(* PLC project BE_Framework BA.project, CODESYS CODESYS V3.5 SP13 Patch 2 *)
(* stored: creationDateTime 2018-12-05T10:06:31.7537871, modificationDateTime 2018-12-03T08:58:43.5869763 *)

PROGRAM LB01_FF1_Analog
VAR
	local:strFan_Analog;
	localGP:strSensor2_Regulator;
	ControlFan: _BE_Fan;
	FbRegulator: _BE_Regulator;
	_BE_Fan2: _BE_Fan_2;
	reset_en: RS;
	AlarmFbAl01: _BE_AlarmAckRequired;
	AlarmFbAl02: _BE_AlarmAckRequired;
	fb_OperationalTime: _BE_OperationalTime;
	ackAl01: BOOL;
	ackAl02: BOOL;
	fanGuardOk: BOOL;
END_VAR
  VAR  (* added by the conversion: wires and edge detectors of the diagram *)
    __49_OUT : REAL;
    _MOVE171_ENO : BOOL;
    _MOVE171_OUT : INT;
    _AND235_OUT : BOOL;
    _AND241_OUT : BOOL;
    _MOVE64_ENO : BOOL;
    _MOVE64_OUT : REAL;
    _MOVE70_ENO : BOOL;
    _MOVE70_OUT : REAL;
    _MOVE151_ENO : BOOL;
    _MOVE151_OUT : ANY;
  END_VAR

(* CFC diagram, written out as Structured Text *)
(* Handling of enable and disable of regulator *)
local := LB01.FF1;
localGP := LB01.GP21;
fanGuardOk := LB01.GP23.V;
local.EnFeedbackError := >(local.SP4, 0);
local.EnThermalError := >(local.SP2, 0);
(* Feedback error *)
local.EnFanGuardError := >(local.SP3, 0);
(* Thermal error *)
(* Regulator *)
_BE_Fan2(AutoStart := LB01.GeneralStart, AutoStartTimeDelay := local.SP1 + 5, BlockAutoStart := false, RunIndication := local.V, EnableFeedbackAlarm := local.EnFeedbackError, FeedbackAlarmTimeDelay := local.SP4, EnableThermicRelayAlarm := local.EnThermalError, ThermicRelayOk := local.ThermoRelay1, ThermicRelayAlarmTimeDelay := local.SP2, EnableFanGuardAlarm := local.EnFanGuardError, FanGuardOk := fanGuardOk, FanGuardAlarmTimeDelay := local.SP3, AlarmIndication := local.AL, AutoReg := local.AUT);
local.CMD := _BE_Fan2.StartSignalOutput;
local.FeedbackError := _BE_Fan2.FeedbackAlarm;
local.ThermalError := _BE_Fan2.ThermicRelayAlarm;
local.FanGuardError := _BE_Fan2.FanGuardAlarm;
(* General Alarm *)
(* Manual control from hardware switches *)
__49_OUT := <(local.OP, 0.5);
(* Manual control from hardware switches *)
local.Symbol := SEL(local.ST2792_M OR local.ST4491_M, SEL(=(_BE_Fan2.Status, 1) AND __49_OUT, _BE_Fan2.Status, 0), SEL(local.ST2792_MCMD AND >(local.ST4491_OPM, 0.5) AND local.ST4491_M, 0, 1));
local.Operating := local.CMD;
(* HMI symbol for the handsymbol in iX *)
local.Symbol_M := 0;
_MOVE171_OUT := MOVE(EN := >(local.AUT, 0) OR local.ST2792_M OR local.ST4491_M, IN := 1, ENO => _MOVE171_ENO);
IF _MOVE171_ENO THEN local.Symbol_M := _MOVE171_OUT; END_IF;
_AND235_OUT := local.ACK AND local.AL01;
IF _AND235_OUT THEN ackAl01 := TRUE; END_IF;
_AND241_OUT := local.ACK AND local.AL02;
IF _AND241_OUT THEN ackAl02 := TRUE; END_IF;
IF true THEN local.ACK := FALSE; END_IF;
AlarmFbAl01(Alarm := local.EnFeedbackError AND local.FeedbackError, InitPulse := SYS_E_AckAlarm, AlarmAck := ackAl01);
local.AL01 := AlarmFbAl01.AlarmActive;
AlarmFbAl02(Alarm := local.EnThermalError AND local.ThermalError, InitPulse := SYS_E_AckAlarm, AlarmAck := ackAl02);
local.AL02 := AlarmFbAl02.AlarmActive;
local.AL := local.AL01 OR local.AL02;
reset_en(SET := local.CMD, RESET1 := NOT local.CMD);
localGP.PID_En := reset_en.Q1;
_MOVE64_OUT := MOVE(EN := NOT local.CMD, IN := 0.0, ENO => _MOVE64_ENO);
IF _MOVE64_ENO THEN local.OP := _MOVE64_OUT; END_IF;
_MOVE70_OUT := MOVE(EN := _MOVE64_ENO, IN := 0.0, ENO => _MOVE70_ENO);
IF _MOVE70_ENO THEN local.OPM := _MOVE70_OUT; END_IF;
localGP.CSP := localGP.SP;
FbRegulator(Enable := localGP.PID_En, SetValue := localGP.CSP, ProcessValue := localGP.PV, DeadBand := localGP.DB, P_Pid := localGP.P, I_Integral := localGP.I, D_Deriv := localGP.D, SampleTime := localGP.SI, OutputValueMax := localGP.MAX1, OutputValueMin := localGP.MIN1, NormalReverse := false, FilterValue := 0.0, Pulse100ms := SYS_Pulse100ms, InitPulse := SYS_InitPulse, Manual := >(local.AUT, 0), ManualAutoFeedback := true, ManualValue := local.OPM, SavedWorkingData := localGP.SavedData, OutputValue := local.OP);
_MOVE151_OUT := MOVE(EN := local.ST4491_M, IN := local.ST4491_OPM, ENO => _MOVE151_ENO);
IF _MOVE151_ENO THEN local.OP := _MOVE151_OUT; END_IF;
fb_OperationalTime(Operating := local.CMD, MinutePulse := SYS_MinutePulse, ResetOperatingTime := local.RST, ResetStarts := local.RST);
local.PV2 := fb_OperationalTime.TotalMinutes;
local.PV1 := fb_OperationalTime.TotalHours;
local.PV3 := fb_OperationalTime.StartsTotal;
LB01.FF1 := local;
LB01.GP21 := localGP;
END_PROGRAM

PROGRAM LB01_Alarm
VAR
	fb_nod1: R_TRIG;
	fb_TON_reset: TON;
	AlarmAcknowledge01: _BE_AlarmAckRemote;
	timerManMode: TON;
	_BE_AlarmAckRemote_0: _BE_AlarmAckRemote;
END_VAR
  VAR  (* added by the conversion: wires and edge detectors of the diagram *)
    _OR55_OUT : INT;
  END_VAR

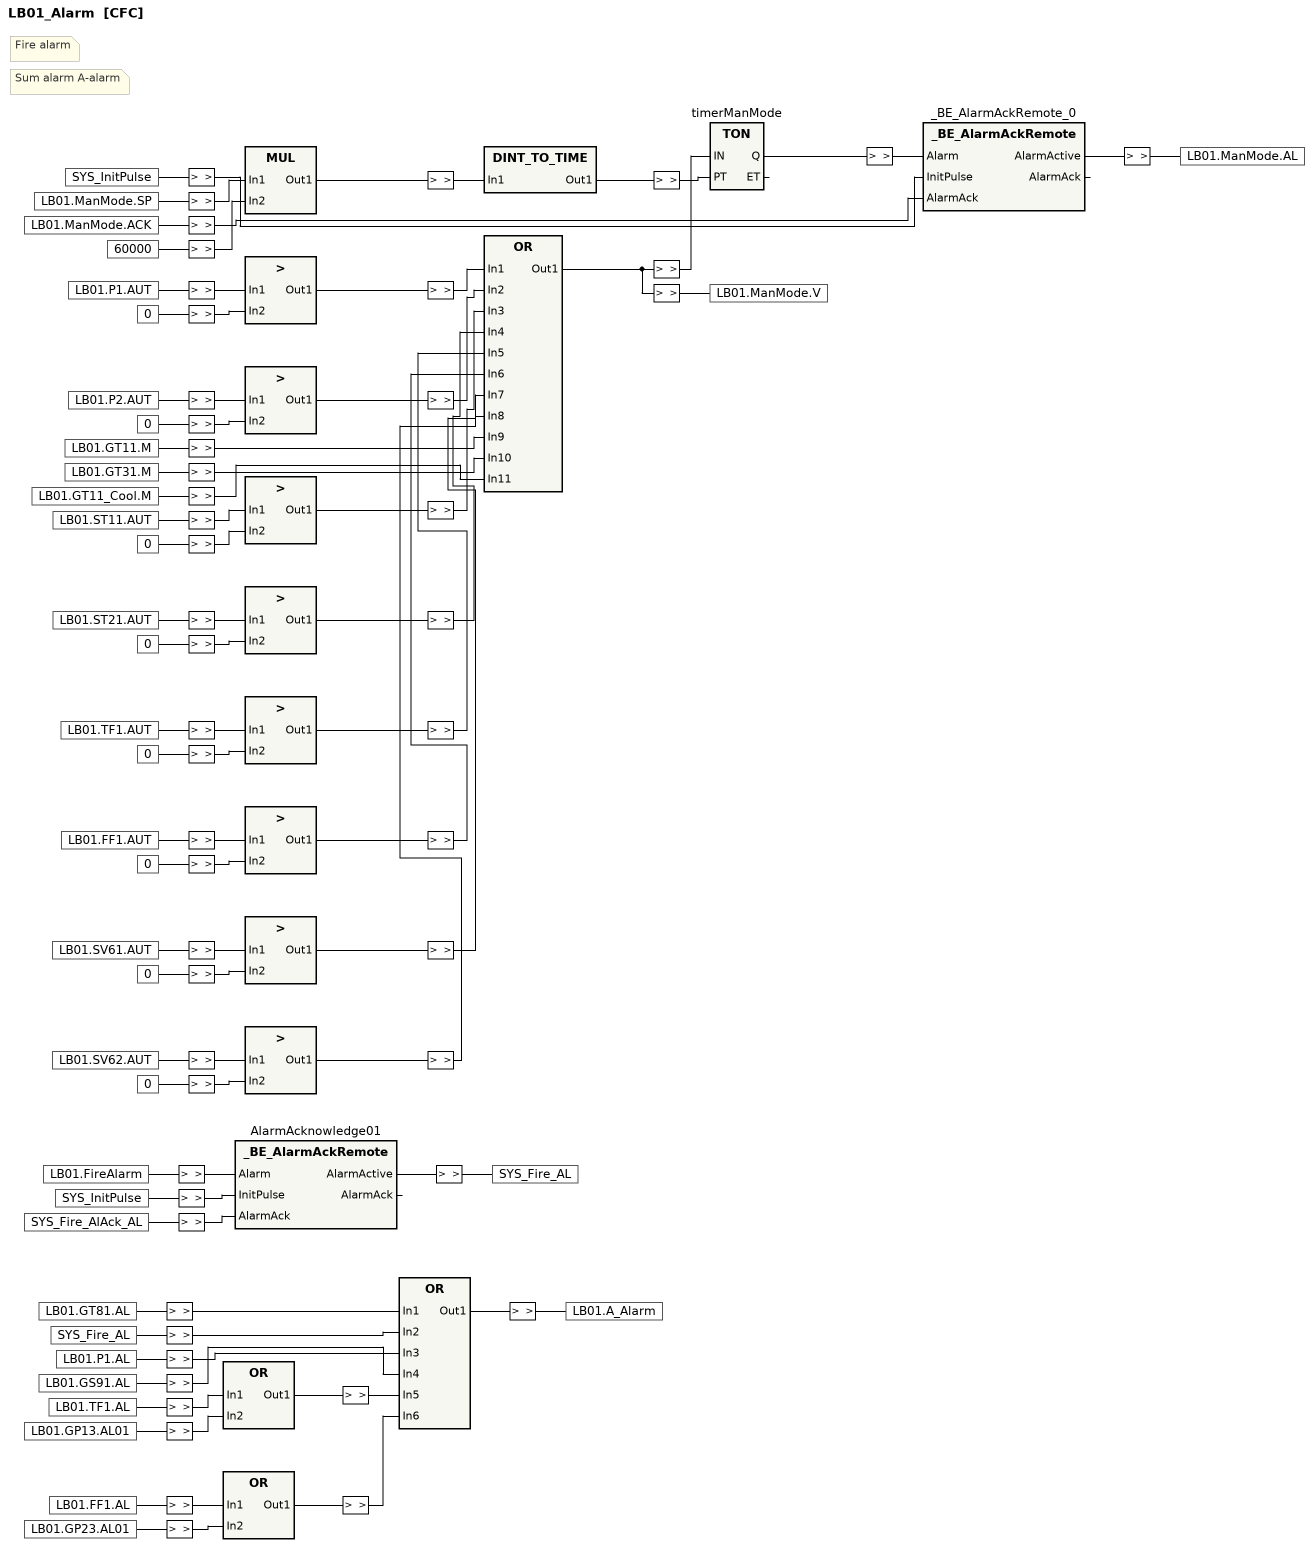
(* CFC diagram, written out as Structured Text *)
(* Fire alarm *)
AlarmAcknowledge01(Alarm := LB01.FireAlarm, InitPulse := SYS_InitPulse, AlarmAck := SYS_Fire_AlAck_AL);
SYS_Fire_AL := AlarmAcknowledge01.AlarmActive;
(* Sum alarm A-alarm *)
LB01.A_Alarm := LB01.GT81.AL OR SYS_Fire_AL OR LB01.P1.AL OR LB01.GS91.AL OR LB01.TF1.AL OR LB01.GP13.AL01 OR LB01.FF1.AL OR LB01.GP23.AL01;
_OR55_OUT := >(LB01.P1.AUT, 0) OR >(LB01.P2.AUT, 0) OR >(LB01.ST11.AUT, 0) OR >(LB01.ST21.AUT, 0) OR >(LB01.TF1.AUT, 0) OR >(LB01.FF1.AUT, 0) OR >(LB01.SV61.AUT, 0) OR >(LB01.SV62.AUT, 0) OR LB01.GT11.M OR LB01.GT31.M OR LB01.GT11_Cool.M;
LB01.ManMode.V := _OR55_OUT;
timerManMode(IN := _OR55_OUT, PT := DINT_TO_TIME(LB01.ManMode.SP * 60000));
_BE_AlarmAckRemote_0(Alarm := timerManMode.Q, InitPulse := SYS_InitPulse, AlarmAck := LB01.ManMode.ACK);
LB01.ManMode.AL := _BE_AlarmAckRemote_0.AlarmActive;
END_PROGRAM
